///EL2008 | 8-channel digital output terminal 24 V DC, 0.5 A
FUNCTION_BLOCK FB_EL2008_v1_00
VAR_INPUT
	En: BOOL;
	bDo_1: BOOL;
	bDo_2: BOOL;
	bDo_3: BOOL;
	bDo_4: BOOL;
	bDo_5: BOOL;
	bDo_6: BOOL;
	bDo_7: BOOL;
	bDo_8: BOOL;
END_VAR
VAR_OUTPUT
	EnO: BOOL;
	bError: BOOL;
END_VAR
VAR
	Channel_1_Output AT %Q*: BOOL;
	Channel_2_Output AT %Q*: BOOL;
	Channel_3_Output AT %Q*: BOOL;
	Channel_4_Output AT %Q*: BOOL;
	Channel_5_Output AT %Q*: BOOL;
	Channel_6_Output AT %Q*: BOOL;
	Channel_7_Output AT %Q*: BOOL;
	Channel_8_Output AT %Q*: BOOL;
	WcState_WcState AT %I*: BOOL;
	InfoData_State AT %I*: UINT;
END_VAR

EnO:=En;

IF En AND (WcState_WcState OR InfoData_State<>16#8) THEN
	bError:=TRUE;
ELSE
	bError:=FALSE;
END_IF

IF En THEN
	IF bError=FALSE THEN
		Channel_1_Output:=bDo_1;
		Channel_2_Output:=bDo_2;
		Channel_3_Output:=bDo_3;
		Channel_4_Output:=bDo_4;
		Channel_5_Output:=bDo_5;
		Channel_6_Output:=bDo_6;
		Channel_7_Output:=bDo_7;
		Channel_8_Output:=bDo_8;
	END_IF
END_IF

END_FUNCTION_BLOCK

(* stored: Version 1.1.0.1, ProductVersion 3.1.4022.6
   POU FB_EL2008_v1_00: Id {801203f0-99cc-4247-be6c-3a0f97b0d87c}, SpecialFunc None *)
